(*
SPDX-FileCopyrightText: © 2026 Oleksandr Tiutyk <trofimich@gmail.com>
SPDX-License-Identifier: MIT
License: https://opensource.org/license/mit
*)

(*!
<summary>
Beckhoff EL3004_EX: Extended 4-channel analog input terminal with diagnostics.
</summary>
<description>
Extends EL3004 with EtherCAT Working Counter, slave state, and CoE mailbox ADS address diagnostics.
When used for I/O, link located fields or their containing buffers to the matching selected PDOs.
The record is not a packed wire buffer; compiler padding is not part of the device specification.
Unlinked/default values do not prove valid I/O. The caller evaluates bus/channel validity before use.
Use one owner task per instance and externally synchronize other access; multi-field snapshots are not atomic.
Copies store data without creating hardware links. Keep borrowed field references valid while consumers are bound.
This passive record performs no validation, synchronization, configuration or protocol advancement.
WcState=TRUE means process-data exchange is invalid. State is acyclic EtherCAT/link information,
not proof of current measurement validity. Link diagnostics to the matching slave InfoData entries.
The selected PDO representation is documented by the base terminal model.
InputToggle signals an input update by changing state; TRUE alone does not mean fresh data.
AdsAddr is acyclic mailbox addressing information, not a measurement-validity indicator.
Select standard status-plus-value PDOs matching the declared Value type; compact value-only PDOs
are outside this model. Configure electrical range and scaling separately on the device.
</description>
*)
TYPE EL3004_EX EXTENDS EL3004 :
STRUCT
	WcState AT %I* : BOOL;
	InputToggle AT %I* : BOOL;
	State AT %I* : UINT;
	AdsAddr AT %I* : Global.AMSADDR;
END_STRUCT
END_TYPE

(* stored: Version 1.1.0.1, ProductVersion 3.1.4026.18
   DUT EL3004_EX: Id {27a478f2-2cfd-4255-ac4c-8543fc825f1e} *)
